FUNCTION_BLOCK FB_CTU_LINT (* counters (up-counter) *)
  (* Standard: 61131-3; Classification: standard counters; Description: Copyright (c) 2011 TU Wien ACIN This program and the accompanying materials are made available under the terms of the Eclipse Public License 2.0 which is available at https://www.eclipse.org/legal/epl-2.0/ SPDX-License-Identifier: EPL-2.0 *)
  (* Version 1.0, 2011-06-21, Monika Wenger, TU Wien ACIN *)
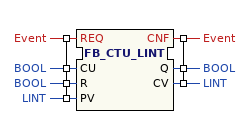
  EVENT_INPUT
    REQ WITH CU, PV, R; (* Service Request *)
  END_EVENT
  EVENT_OUTPUT
    CNF WITH Q, CV; (* Confirmation of Requested Service *)
  END_EVENT
  VAR_INPUT
    CU : BOOL; (* Count up (Rising Edge Detection) *)
    R : BOOL; (* Reset *)
    PV : LINT; (* Preset value *)
  END_VAR
  VAR_OUTPUT
    Q : BOOL; (* Output *)
    CV : LINT; (* Count value *)
  END_VAR
  (* Service APPLICATION/RESOURCE: counters (up-counter) *)
END_FUNCTION_BLOCK
